KUKA KRL program: Zivid_cam.src, Zivid_cam.dat

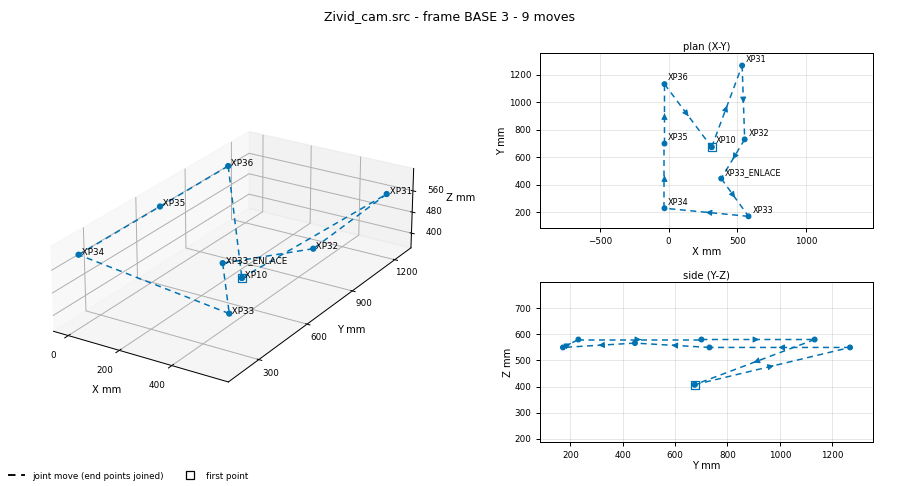
[picture p0: tool path of Zivid_cam.src in frame BASE 3, 9 of 13 moves have a stored position in this frame; points joined in program order, loops and branches not executed]
--- Zivid_cam.src ---
&ACCESS RVP
&REL 48
&COMMENT COGER ST121 RACK AZUL
&PARAM EDITMASK = *
&PARAM TEMPLATE = C:\KRC\Roboter\Template\vorgabe
&PARAM DISKPATH = KRC:\R1\Program\MAFELEC
DEF Zivid_cam( )
;FOLD INI;%{PE}
  ;FOLD BASISTECH INI
    GLOBAL INTERRUPT DECL 3 WHEN $STOPMESS==TRUE DO IR_STOPM ( )
    INTERRUPT ON 3
    BAS (#INITMOV,0 )
  ;ENDFOLD (BASISTECH INI)
;FOLD SPOTTECH INI
USERSPOT(#INIT)
;ENDFOLD (SPOTTECH INI)
;FOLD GRIPPERTECH INI
USER_GRP(0,DUMMY,DUMMY,GDEFAULT)
;ENDFOLD (GRIPPERTECH INI)
;FOLD USER INI
INTERRUPT DECL 26 WHEN I_121R1S102 OR I_121R1S202 DO PARO_RAPIDO ()
INTERRUPT DECL 27 WHEN I_121R1S302 OR I_121R1S402 DO PARO_RAPIDO ()

    ;Make your modifications here

  ;ENDFOLD (USER INI)
;ENDFOLD (INI)
;################################################
; PROYECTO: ZIVID PLANTA DE BATERIAS
; ROBOT: 121_R1 TERMINATOR
; PROGRAMA: Zivid_cam EN ST121
;           PALETA A INSPECCION
; CREADO POR: Borja Carrion
; FECHA: 30-DICIEMBRE-2023
;################################################

Empujador(1,"R",FALSE)
Empujador(2,"R",FALSE)

;FOLD PTP HOME Vel=100 % DEFAULT;%{PE}%R 8.3.48,%MKUKATPBASIS,%CMOVE,%VPTP,%P 1:PTP, 2:HOME, 3:, 5:100, 7:DEFAULT
$BWDSTART=FALSE
PDAT_ACT=PDEFAULT
FDAT_ACT=FHOME
BAS(#PTP_PARAMS,100)
$H_POS=XHOME
PTP XHOME
;ENDFOLD
; FOLD ESPERA CONFIRMACION ENTRADA INSPECCION
WAIT FOR I_ST121_INSPECCION
; ENDFOLD

;FOLD PTP POS_ESPERA_ST121 Vel=100 % H Tool[9]:T_Gripper1_Vacio Base[0];%{PE}%R 8.3.48,%MKUKATPBASIS,%CMOVE,%VPTP,%P 1:PTP, 2:POS_ESPERA_ST121, 3:, 5:100, 7:H
$BWDSTART=FALSE
PDAT_ACT=PH
FDAT_ACT=FPOS_ESPERA_ST121
BAS(#PTP_PARAMS,100)
PTP XPOS_ESPERA_ST121
;ENDFOLD

; FOLD ESPERA CONFIRMACION ENTRADA INSPECCION
WAIT FOR I_ST121_INSPECCION
; ENDFOLD

; FOLD CONTROL DE ELEMENTOS MECANICOS EN REPOSO
;CONTROL DE AUSENCIA DE PIEZA EN GRIPPER
IF I_121R1S1000 THEN
HALT
ENDIF

;CONTROL APERTURA GRIPPER

IF (I_121R1S131B==FALSE) OR (I_121R1S132B==FALSE) OR (I_121R1S133B==FALSE) OR (I_121R1S134B==FALSE) THEN
Pines("R")
ENDIF

Empujador(1,"R",TRUE)
Empujador(2,"R",TRUE)
; ENDFOLD

;FOLD PTP P10 CONT Vel=100 % M Tool[9]:T_Gripper1_Vacio Base[3]:ST121;%{PE}%R 8.3.48,%MKUKATPBASIS,%CMOVE,%VPTP,%P 1:PTP, 2:P10, 3:C_DIS, 5:100, 7:M
$BWDSTART=FALSE
PDAT_ACT=PM
FDAT_ACT=FP10
BAS(#PTP_PARAMS,100)
PTP XP10 C_DIS
;ENDFOLD

; POSICIONES FOTOS CAMARA ZIVID

; FOTO 1 CAMARA ZIVID
;FOLD PTP P31 CONT Vel=50 % M Tool[9]:T_Gripper1_Vacio Base[3]:ST121;%{PE}%R 8.3.48,%MKUKATPBASIS,%CMOVE,%VPTP,%P 1:PTP, 2:P31, 3:C_DIS, 5:50, 7:M
$BWDSTART=FALSE
PDAT_ACT=PM
FDAT_ACT=FP31
BAS(#PTP_PARAMS,50)
PTP XP31 C_DIS
;ENDFOLD
WAIT SEC 0.2

; FOTO 2 CAMARA ZIVID
;FOLD PTP P32 CONT Vel=50 % M Tool[9]:T_Gripper1_Vacio Base[3]:ST121;%{PE}%R 8.3.48,%MKUKATPBASIS,%CMOVE,%VPTP,%P 1:PTP, 2:P32, 3:C_DIS, 5:50, 7:M
$BWDSTART=FALSE
PDAT_ACT=PM
FDAT_ACT=FP32
BAS(#PTP_PARAMS,50)
PTP XP32 C_DIS
;ENDFOLD
WAIT SEC 0.2

;FOLD PTP P33_ENLACE CONT Vel=50 % H Tool[9]:T_Gripper1_Vacio Base[3]:ST121;%{PE}%R 8.3.48,%MKUKATPBASIS,%CMOVE,%VPTP,%P 1:PTP, 2:P33_ENLACE, 3:C_DIS, 5:50, 7:H
$BWDSTART=FALSE
PDAT_ACT=PH
FDAT_ACT=FP33_ENLACE
BAS(#PTP_PARAMS,50)
PTP XP33_ENLACE C_DIS
;ENDFOLD
; FOTO 3 CAMARA ZIVID
;FOLD PTP P33 CONT Vel=50 % M Tool[9]:T_Gripper1_Vacio Base[3]:ST121;%{PE}%R 8.3.48,%MKUKATPBASIS,%CMOVE,%VPTP,%P 1:PTP, 2:P33, 3:C_DIS, 5:50, 7:M
$BWDSTART=FALSE
PDAT_ACT=PM
FDAT_ACT=FP33
BAS(#PTP_PARAMS,50)
PTP XP33 C_DIS
;ENDFOLD
WAIT SEC 0.2

; FOTO 4 CAMARA ZIVID
;FOLD PTP P34 CONT Vel=50 % M Tool[9]:T_Gripper1_Vacio Base[3]:ST121;%{PE}%R 8.3.48,%MKUKATPBASIS,%CMOVE,%VPTP,%P 1:PTP, 2:P34, 3:C_DIS, 5:50, 7:M
$BWDSTART=FALSE
PDAT_ACT=PM
FDAT_ACT=FP34
BAS(#PTP_PARAMS,50)
PTP XP34 C_DIS
;ENDFOLD
WAIT SEC 0.2

; FOTO 5 CAMARA ZIVID
;FOLD PTP P35 CONT Vel=50 % M Tool[9]:T_Gripper1_Vacio Base[3]:ST121;%{PE}%R 8.3.48,%MKUKATPBASIS,%CMOVE,%VPTP,%P 1:PTP, 2:P35, 3:C_DIS, 5:50, 7:M
$BWDSTART=FALSE
PDAT_ACT=PM
FDAT_ACT=FP35
BAS(#PTP_PARAMS,50)
PTP XP35 C_DIS
;ENDFOLD
WAIT SEC 0.2

; FOTO 6 CAMARA ZIVID
;FOLD PTP P36 CONT Vel=50 % M Tool[9]:T_Gripper1_Vacio Base[3]:ST121;%{PE}%R 8.3.48,%MKUKATPBASIS,%CMOVE,%VPTP,%P 1:PTP, 2:P36, 3:C_DIS, 5:50, 7:M
$BWDSTART=FALSE
PDAT_ACT=PM
FDAT_ACT=FP36
BAS(#PTP_PARAMS,50)
PTP XP36 C_DIS
;ENDFOLD
WAIT SEC 0.2

;FOLD PTP POS_SOBRE_ST121 Vel=50 % H Tool[9]:T_Gripper1_Vacio Base[3]:ST121;%{PE}%R 8.3.48,%MKUKATPBASIS,%CMOVE,%VPTP,%P 1:PTP, 2:POS_SOBRE_ST121, 3:, 5:50, 7:H
$BWDSTART=FALSE
PDAT_ACT=PH
FDAT_ACT=FPOS_SOBRE_ST121
BAS(#PTP_PARAMS,50)
PTP XPOS_SOBRE_ST121
;ENDFOLD


;POSICION AREA 3 LIBRE
;FOLD PTP POS_ESPERA_ST122 Vel=100 % H Tool[9]:T_Gripper1_Vacio Base[0];%{PE}%R 8.3.48,%MKUKATPBASIS,%CMOVE,%VPTP,%P 1:PTP, 2:POS_ESPERA_ST122, 3:, 5:100, 7:H
$BWDSTART=FALSE
PDAT_ACT=PH
FDAT_ACT=FPOS_ESPERA_ST122
BAS(#PTP_PARAMS,100)
PTP XPOS_ESPERA_ST122
;ENDFOLD

;LIBERA AREA 3, TRANSPORTE BATERIAS
O_AREL_3=TRUE


;FOLD PTP HOME Vel=100 % DEFAULT;%{PE}%R 8.3.48,%MKUKATPBASIS,%CMOVE,%VPTP,%P 1:PTP, 2:HOME, 3:, 5:100, 7:DEFAULT
$BWDSTART=FALSE
PDAT_ACT=PDEFAULT
FDAT_ACT=FHOME
BAS(#PTP_PARAMS,100)
$H_POS=XHOME
PTP XHOME
;ENDFOLD

END
DEF PARO_RAPIDO ()
BRAKE F
END

--- Zivid_cam.dat ---
&ACCESS RVP
&REL 48
&COMMENT COGER ST121 RACK AZUL
&PARAM EDITMASK = *
&PARAM TEMPLATE = C:\KRC\Roboter\Template\vorgabe
&PARAM DISKPATH = KRC:\R1\Program\MAFELEC
DEFDAT  Zivid_cam
;FOLD EXTERNAL DECLARATIONS;%{PE}%MKUKATPBASIS,%CEXT,%VCOMMON,%P
;FOLD GRIPPERTECH EXT
EXT  H50 (INT  :IN,INT  :IN,INT  :IN,GRP_TYP  :IN )
;ENDFOLD (GRIPPERTECH EXT)
;FOLD SPOTTECH EXT
EXT  USERSPOT (S_COMMAND  :IN,SPOT_TYPE  :IN )
;ENDFOLD (SPOTTECH EXT)
;FOLD BASISTECH EXT;%{PE}%MKUKATPBASIS,%CEXT,%VEXT,%P
EXT  BAS (BAS_COMMAND  :IN,REAL  :IN )
DECL INT SUCCESS
;ENDFOLD (BASISTECH EXT)
;FOLD USER EXT;%{E}%MKUKATPUSER,%CEXT,%VEXT,%P
;Make your modifications here

;ENDFOLD (USER EXT)
;ENDFOLD (EXTERNAL DECLARATIONS)
DECL BASIS_SUGG_T LAST_BASIS={POINT1[] "P33_ENLACE              ",POINT2[] "P33_ENLACE              ",CP_PARAMS[] "M                       ",PTP_PARAMS[] "H                       ",CONT[] "C_DIS                   ",CP_VEL[] "0.2                     ",PTP_VEL[] "50                      ",SYNC_PARAMS[] "SYNCDAT                 ",SPL_NAME[] "S0                      ",A_PARAMS[] "ADAT0                   "}
DECL PDAT PH={VEL 100.000,ACC 100.000,APO_DIST 100.000,APO_MODE #CDIS,GEAR_JERK 50.0000,EXAX_IGN 0}
DECL E6POS XP10={X 312.450226,Y 675.070,Z 407.579834,A -0.219463497,B -0.287549138,C -179.748962,S 2,T 42,E1 0.0,E2 0.0,E3 0.0,E4 0.0,E5 0.0,E6 0.0}
DECL FDAT FP10={TOOL_NO 9,BASE_NO 3,IPO_FRAME #BASE,POINT2[] " ",TQ_STATE FALSE}
DECL E6POS XP20={X 312.450226,Y 675.070,Z 73.4258270,A -0.219463497,B -0.287549138,C -179.748962,S 2,T 42,E1 0.0,E2 0.0,E3 0.0,E4 0.0,E5 0.0,E6 0.0}
DECL FDAT FP20={TOOL_NO 9,BASE_NO 3,IPO_FRAME #BASE,POINT2[] " ",TQ_STATE FALSE}
DECL E6POS XPOS_COGER_ST121={X 364.233917,Y 680.820,Z 35.4071388,A -0.219463244,B -0.287549198,C -179.748962,S 2,T 42,E1 0.0,E2 0.0,E3 0.0,E4 0.0,E5 0.0,E6 0.0}
DECL FDAT FPos_Coger_ST121={TOOL_NO 9,BASE_NO 3,IPO_FRAME #BASE,POINT2[] " ",TQ_STATE FALSE}
DECL PDAT PM={VEL 100.000,ACC 50.0000,APO_DIST 50.0000,APO_MODE #CDIS,GEAR_JERK 50.0000,EXAX_IGN 0}
DECL E6POS XPOS_ESPERA_ST121={X 1597.05444,Y -395.116150,Z 1941.31274,A -176.307449,B 30.3077869,C -171.065643,S 2,T 10,E1 0.0,E2 0.0,E3 0.0,E4 0.0,E5 0.0,E6 0.0}
DECL FDAT FPOS_ESPERA_ST121={TOOL_NO 9,BASE_NO 0,IPO_FRAME #BASE,POINT2[] " ",TQ_STATE FALSE}
DECL LDAT LM={VEL 2.00000,ACC 25.0000,APO_DIST 100.000,APO_FAC 50.0000,AXIS_VEL 100.000,AXIS_ACC 100.000,ORI_TYP #VAR,CIRC_TYP #BASE,JERK_FAC 50.0000,GEAR_JERK 50.0000,EXAX_IGN 0}
DECL E6POS XPOS_SOBRE_ST121={X 312.450226,Y 675.070,Z 407.579834,A -0.219463497,B -0.287549138,C -179.748962,S 2,T 42,E1 0.0,E2 0.0,E3 0.0,E4 0.0,E5 0.0,E6 0.0}
DECL FDAT FPOS_SOBRE_ST121={TOOL_NO 9,BASE_NO 3,IPO_FRAME #BASE,POINT2[] " ",TQ_STATE FALSE}
DECL E6POS XPOS_SOBRE_ST122={X 1790.32410,Y 1.34322268E-13,Z 1909.62585,A -180.000,B 89.9853210,C -180.000,S 2,T 3,E1 0.0,E2 0.0,E3 0.0,E4 0.0,E5 0.0,E6 0.0}
DECL FDAT FPOS_SOBRE_ST122={TOOL_NO 9,BASE_NO 3,IPO_FRAME #BASE,POINT2[] " ",TQ_STATE FALSE}
DECL E6POS XP30={X 158.918106,Y 1091.44617,Z 654.405884,A 42.3399849,B -0.235063374,C -179.753174,S 2,T 42,E1 0.0,E2 0.0,E3 0.0,E4 0.0,E5 0.0,E6 0.0}
DECL FDAT FP30={TOOL_NO 11,BASE_NO 3,IPO_FRAME #BASE,POINT2[] " ",TQ_STATE FALSE}
DECL E6POS XP40={X -0.0319372341,Y -2.62910700,Z -362.053223,A -0.00123304490,B -0.0257057231,C 0.00384289422,S 2,T 10,E1 0.0,E2 0.0,E3 0.0,E4 0.0,E5 0.0,E6 0.0}
DECL FDAT FP40={TOOL_NO 11,BASE_NO 3,IPO_FRAME #BASE,POINT2[] " ",TQ_STATE FALSE}
DECL E6POS XPOS_AREA_3_LIBRE={X 1597.05457,Y -395.116180,Z 1941.31274,A -176.307449,B 30.3077888,C -171.065643,S 2,T 10,E1 0.0,E2 0.0,E3 0.0,E4 0.0,E5 0.0,E6 0.0}
DECL FDAT FPOS_AREA_3_LIBRE={TOOL_NO 9,BASE_NO 3,IPO_FRAME #BASE,POINT2[] " ",TQ_STATE FALSE}
DECL GRP_SUGG_T LAST_GRP={NUMBER[] "1                       ",STATE[] "1                       ",PARAMS[] "GDAT0                   "}
DECL LDAT LL={VEL 2.00000,ACC 25.0000,APO_DIST 100.000,APO_FAC 50.0000,AXIS_VEL 100.000,AXIS_ACC 100.000,ORI_TYP #VAR,CIRC_TYP #BASE,JERK_FAC 50.0000,GEAR_JERK 50.0000,EXAX_IGN 0}
DECL PDAT PL={VEL 100.000,ACC 25.0000,APO_DIST 50.0000,APO_MODE #CDIS,GEAR_JERK 50.0000,EXAX_IGN 0}
DECL E6POS XP0={X 364.480164,Y 681.182129,Z 388.540192,A -0.219463348,B -0.287549168,C -179.748962,S 2,T 42,E1 0.0,E2 0.0,E3 0.0,E4 0.0,E5 0.0,E6 0.0}
DECL FDAT FP0={TOOL_NO 9,BASE_NO 3,IPO_FRAME #BASE,POINT2[] " ",TQ_STATE FALSE}
DECL E6POS XP1={X 364.233917,Y 677.270142,Z 82.2082901,A -0.219467312,B -0.287552059,C -179.748962,S 2,T 42,E1 0.0,E2 0.0,E3 0.0,E4 0.0,E5 0.0,E6 0.0}
DECL FDAT FP1={TOOL_NO 9,BASE_NO 3,IPO_FRAME #BASE,POINT2[] " ",TQ_STATE FALSE}
DECL E6POS XPos_Coger_Verde_ST121={X 364.233917,Y 680.820,Z 35.4071388,A -0.219467372,B -0.287552029,C -179.748962,S 2,T 42,E1 0.0,E2 0.0,E3 0.0,E4 0.0,E5 0.0,E6 0.0}
DECL FDAT FPos_Coger_Verde_ST121={TOOL_NO 9,BASE_NO 3,IPO_FRAME #BASE,POINT2[] " ",TQ_STATE FALSE}
DECL E6POS XCOGER_ST121_INSP={X 312.450226,Y 675.070,Z 31.2908478,A -0.219463453,B -0.287549138,C -179.748962,S 2,T 42,E1 0.0,E2 0.0,E3 0.0,E4 0.0,E5 0.0,E6 0.0}
DECL FDAT FCoger_ST121_INSP={TOOL_NO 9,BASE_NO 3,IPO_FRAME #BASE,POINT2[] " ",TQ_STATE FALSE}
DECL E6POS XPOS_ESPERA_ST122={X 1597.05444,Y -395.116150,Z 1941.31274,A -176.307449,B 30.3077869,C -171.065643,S 2,T 10,E1 0.0,E2 0.0,E3 0.0,E4 0.0,E5 0.0,E6 0.0}
DECL FDAT FPOS_ESPERA_ST122={TOOL_NO 9,BASE_NO 0,IPO_FRAME #BASE,POINT2[] " ",TQ_STATE FALSE}
DECL E6POS XP31={X 534.243774,Y 1268.12231,Z 549.593567,A -0.478079498,B -8.25281906,C -179.458313,S 2,T 43,E1 0.0,E2 0.0,E3 0.0,E4 0.0,E5 0.0,E6 0.0}
DECL FDAT FP31={TOOL_NO 9,BASE_NO 3,IPO_FRAME #BASE,POINT2[] " ",TQ_STATE FALSE}
DECL E6POS XP32={X 552.691772,Y 731.378,Z 549.580139,A -0.478093654,B -8.25281811,C -179.458313,S 2,T 42,E1 0.0,E2 0.0,E3 0.0,E4 0.0,E5 0.0,E6 0.0}
DECL FDAT FP32={TOOL_NO 9,BASE_NO 3,IPO_FRAME #BASE,POINT2[] " ",TQ_STATE FALSE}
DECL E6POS XP33={X 580.570618,Y 171.789917,Z 549.577698,A -10.8831120,B -8.25385761,C -179.458237,S 2,T 42,E1 0.0,E2 0.0,E3 0.0,E4 0.0,E5 0.0,E6 0.0}
DECL FDAT FP33={TOOL_NO 9,BASE_NO 3,IPO_FRAME #BASE,POINT2[] " ",TQ_STATE FALSE}
DECL E6POS XP34={X -30.1993256,Y 230.685913,Z 579.868530,A 1.90679479,B -4.28973961,C -179.402,S 2,T 42,E1 0.0,E2 0.0,E3 0.0,E4 0.0,E5 0.0,E6 0.0}
DECL FDAT FP34={TOOL_NO 9,BASE_NO 3,IPO_FRAME #BASE,POINT2[] " ",TQ_STATE FALSE}
DECL E6POS XP35={X -30.1993980,Y 700.609619,Z 579.868530,A 1.90679491,B -4.28973961,C -179.402,S 2,T 42,E1 0.0,E2 0.0,E3 0.0,E4 0.0,E5 0.0,E6 0.0}
DECL FDAT FP35={TOOL_NO 9,BASE_NO 3,IPO_FRAME #BASE,POINT2[] " ",TQ_STATE FALSE}
DECL E6POS XP36={X -30.2382946,Y 1133.01782,Z 579.867065,A 1.90679693,B -4.28984737,C -179.401978,S 2,T 42,E1 0.0,E2 0.0,E3 0.0,E4 0.0,E5 0.0,E6 0.0}
DECL FDAT FP36={TOOL_NO 9,BASE_NO 3,IPO_FRAME #BASE,POINT2[] " ",TQ_STATE FALSE}
DECL E6POS XP33_ENLACE={X 382.159821,Y 446.730743,Z 566.171936,A -5.97425365,B -8.25511932,C -179.447327,S 2,T 42,E1 0.0,E2 0.0,E3 0.0,E4 0.0,E5 0.0,E6 0.0}
DECL FDAT FP33_ENLACE={TOOL_NO 9,BASE_NO 3,IPO_FRAME #BASE,POINT2[] " ",TQ_STATE FALSE}
ENDDAT
